(* PLC project Sin nombre, Desconocido Sin nombre 1 *)
(* stored: creationDateTime 2025-05-29T14:31:43, modificationDateTime 2025-05-29T18:50:45 *)

PROGRAM Memorias
  VAR
    I_NA0 AT %IX0.0 : BOOL;  (* D17 - I0.0 *)
    I_NA1 AT %IX0.1 : BOOL;  (* D18 - I0.1 *)
  END_VAR
  VAR
    M0 : BOOL;
  END_VAR
  VAR
    Q_NA AT %QX0.1 : BOOL;  (* D2 - Q0.1 *)
  END_VAR

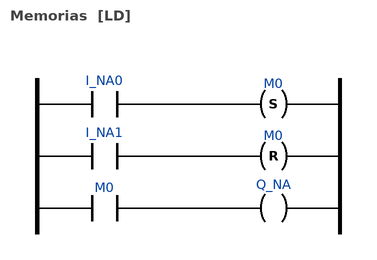
(* LD diagram, written out as Structured Text *)
Q_NA := M0;
IF I_NA1 THEN M0 := FALSE; END_IF;
IF I_NA0 THEN M0 := TRUE; END_IF;
END_PROGRAM

CONFIGURATION Config0
  RESOURCE Res0 ON PLC
    TASK task0(INTERVAL := T#20ms, PRIORITY := 0);
    PROGRAM instance0 WITH task0 : Memorias;
  END_RESOURCE
END_CONFIGURATION
